RoboDK station: conveyor.rdk

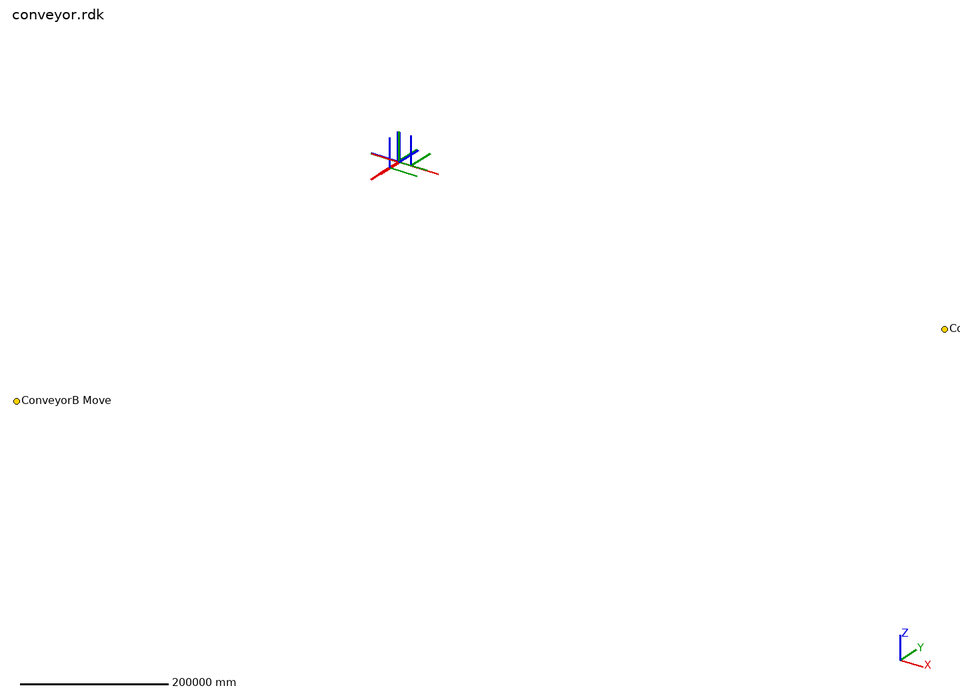
[picture v0: the station drawn from its stored meshes, robots at their saved joint values, targets as dots, program paths as lines]
Station conveyor (saved by RoboDK 6.0.4). Poses are relative to the parent item; angles as X-Y-Z fixed-axis rotations.
Station parameters (name, value as stored): SICK WL4S Laser Sensor, 1
  - notes Description: <!DOCTYPE HTML PUBLIC "-//W3C//DTD HTML 4.0//EN" "http://www.w3.org/TR/REC-html40/strict.dtd">
<html><head><meta name="qrichtext" content="1" /><style type="text/css">
p, li { white-space: pre-wrap; }
</style></head><body style=" font-family:'MS Shell Dlg 2'; font-size:8.25pt; font-weight:400; font-style:normal;">
<p style=" margin-top:0px; margin-bottom:0px; margin-left:0px; margin-right:0px; -qt-block-indent:0; text-indent:0px;">This example showcase how you can use the event instruction to simulation object spawning and conveyor movements.<br /><br />To use this feature, right click on the program -&gt; Add instruction -&gt; Simulation Event Instruction -&gt; Actions<br /><br />All actions you can simulate are the following : <br />Attach object <br />Detach object<br />Show object/tool</p>
<p style=" margin-top:0px; margin-bottom:0px; margin-left:0px; margin-right:0px; -qt-block-indent:0; text-indent:0px;">Hide object/hive</p>
<p style=" margin-top:0px; margin-bottom:0px; margin-left:0px; margin-right:0px; -qt-block-indent:0; text-indent:0px;">Set object position (absolute)<br />Set object position (relative)</p>
<p style=" margin-top:0px; margin-bottom:0px; margin-left:0px; margin-right:0px; -qt-block-indent:0; text-indent:0px;">Set joints home<br />Move conveyor</p>
<p style=" margin-top:0px; margin-bottom:0px; margin-left:0px; margin-right:0px; -qt-block-indent:0; text-indent:0px;">Create object</p>
<p style=" margin-top:0px; margin-bottom:0px; margin-left:0px; margin-
  - frame WCS at (0, 0, 0) mm
    - frame ABB CRB 1300-7/1.4 Base at (1424.15, -838.06, 0) mm, rotated rx 0 ry 0 rz 90 deg
      - robot ABB CRB 1300-7/1.4: 6 axes
          modified DH rows (alpha deg, a mm, theta deg, d mm): 0, 0, 0, 544; -90, 150, -90, 0; 0, 575, 0, 0; -90, 40, 0, 675; 90, 0, 0, 0; -90, 0, 180, 90
          joint limits [-180, -95, -210, -230, -130, -242] to [180, 155, 69, 230, 130, 242]; home [0, 0, 0, 0, 0, 0]; saved at [0, 0, 0, 0, 0, 0]
    - frame Reference Box Frame at (60, 290, 366.5) mm
      - object Box at (0, 0, 0) mm, size 252 x 305.4 x 216.7 mm, geometry from UUID&
    - frame ConveyorA Base at (0, 0, 0) mm
      - robot ConveyorA: 1 axes
          modified DH rows (alpha deg, a mm, theta deg, d mm): 0, 0, 0, 0 linear
          base shift (0, 0, 0) mm, rotated rx 0 ry 90 rz 0 deg
          joint limits [-900000] to [900000]; home [0]; saved at [22355]
        - frame ConveyorA Move Ref at (0, 0, 0) mm
          - object Box at (-20407, 290, 0) mm, size 252 x 305.4 x 216.7 mm, geometry from UUID&
          - object Box at (-21111, 290, 0) mm, size 252 x 305.4 x 216.7 mm, geometry from UUID&
          - object Box at (-21817, 290, 0) mm, size 252 x 305.4 x 216.7 mm, geometry from UUID&
      - target ConveyorA Move (joint target) at (900000, 0, 366.5) mm; joints [900000] of ConveyorA
      - frame Laser Sensor A at (1579.34, 686.74, 443.91) mm, rotated rx 90 ry 0 rz -90 deg
        - object Laser Sensor A at (0, 0, 0) mm, size 683.3 x 45.2 x 12.5 mm, geometry from UUID&
    - frame ConveyorB 2m Base at (2170, 690, 0) mm, rotated rx 0 ry 0 rz -90 deg
      - robot ConveyorB: 1 axes
          modified DH rows (alpha deg, a mm, theta deg, d mm): 0, 0, 0, 0 linear
          base shift (0, 0, 0) mm, rotated rx 0 ry 90 rz 0 deg
          joint limits [-900000] to [900000]; home [0]; saved at [22348]
        - frame ConveyorB Move Ref at (0, 0, 0) mm
          - object Box at (-20951, 193, 0) mm, rotated rx 0 ry 0 rz 90 deg, size 252 x 305.4 x 216.7 mm, geometry from UUID&
          - object Box at (-21655, 192, 0) mm, rotated rx 0 ry 0 rz 90 deg, size 252 x 305.4 x 216.7 mm, geometry from UUID&
      - target ConveyorB Move (joint target) at (900000, 0, 366.5) mm; joints [900000] of ConveyorB
      - frame Laser Sensor B at (1702.6, 686.74, 443.91) mm, rotated rx 90 ry 0 rz -90 deg
        - object Laser Sensor B at (0, 0, 0) mm, size 683.3 x 45.2 x 12.5 mm, geometry from UUID&
      - object Swap conveyor trigger at (395.25, 361.54, 421.76) mm, size 100 x 100 x 100 mm, geometry from UUID&
  - program MainSimulation (7 instructions, listed below)
  - program ResetSimulation (3 instructions, listed below)
  - program BoxDeleterB (1 instructions, listed below)
  - program ConveyorSwap (1 instructions, listed below)
  - program ConveyorMoveA (1 instructions, listed below)
  - program ConveyorMoveB (1 instructions, listed below)
  - program BoxFeeder (2 instructions, listed below)

--- program MainSimulation (robot ConveyorA) ---
  Call ResetSimulation
  Run BoxDeleterA
  Run BoxDeleterB
  Run ConveyorSwap
  Run ConveyorMoveA
  Run ConveyorMoveB
  Run BoxFeeder

--- program ResetSimulation (robot ConveyorA) ---
  Home ConveyorA
  Home ConveyorB
  Remove all Box

--- program BoxDeleterB ---
  Wait & Remove-Laser Sensor B

--- program ConveyorSwap ---
  Wait & Move-Swap conveyor trigger

--- program ConveyorMoveA (robot ConveyorA) ---
  MoveJ (Conveyor Move) -> target ConveyorA Move

--- program ConveyorMoveB (robot ConveyorB) ---
  MoveJ (ConveyorB Move)

--- program BoxFeeder ---
  Feed Reference Box
  Pause 7.0 s
